Fanuc KAREL source: kt00294.KL

-- PROVISIONAL review KL for V1013-1; original PC SHA256 636bf92633a810cad67a8d4bb2511642772355719401841d72fb21d9791b37cb
-- Incomplete behavior may be omitted. Consult companion uncertainty JSON. Do not deploy.
PROGRAM KT00294
%NOLOCKGROUP
VAR
  I1 : INTEGER
  R2 : REAL
  OUT : BOOLEAN
BEGIN
  -- UNRESOLVED_PC offsets 5-16; opcodes 2E,23
  -- UNRESOLVED_PC offsets 21-32; opcodes 2E,23
  -- UNRESOLVED_PC offsets 37-58; opcodes 21,21,29,64,6E,23
  -- UNRESOLVED_PC offsets 63-67; opcodes 7F
END KT00294
